// TIA Portal V21 export
DATA_BLOCK "MODBUS"   // DB99
{ S7_Optimized_Access := 'FALSE' }
   VAR
      "WRITE CONVEYOR" : Struct
         RUN : Int;
         SPEED : Int;
      END_STRUCT;
      "WRITE TURBINE" : Struct
         RUN : Int;
         SPEED : Int;
      END_STRUCT;
      "WRITE TURBINE2" : Struct
         RUN : Int;
         SPEED : Int;
      END_STRUCT;
      READ : Struct
         CONVEYOR : Int;
         TURBINE : Int;
         TURBINE2 : Int;
      END_STRUCT;
      "CONVEYOR STATUS" : Struct
         "W.DONE" : Bool;
         "W.ERROR" : Bool;
         "W.BUSY" : Bool;
         "W.STATUS" : Word;
         "R.DONE" : Bool;
         "R.ERROR" : Bool;
         "R.BUSY" : Bool;
         "R.STATUS" : Word;
      END_STRUCT;
      "TURBINE STATUS" : Struct
         "W.DONE" : Bool;
         "W.ERROR" : Bool;
         "W.BUSY" : Bool;
         "W.STATUS" : Word;
         "R.DONE" : Bool;
         "R.ERROR" : Bool;
         "R.BUSY" : Bool;
         "R.STATUS" : Word;
      END_STRUCT;
      "TURBINE2 STATUS" : Struct
         "W.DONE" : Bool;
         "W.ERROR" : Bool;
         "W.BUSY" : Bool;
         "W.STATUS" : Word;
         "R.DONE" : Bool;
         "R.ERROR" : Bool;
         "R.BUSY" : Bool;
         "R.STATUS" : Word;
      END_STRUCT;
      NOMX1 : Real;
      NOMX2 : Real;
      "NOM 3" : Real;
      "NOM 4" : Real;
      NOM5 : Real;
      NOM6 : Real;
      "READ TURB" : Struct
         "TURB1 READY" : Bool;
      END_STRUCT;
      "READ DRM" : Array[0..10] of Int;
   END_VAR
BEGIN
END_DATA_BLOCK
